// TIA Portal V20 export
TYPE "typeGlobalClockMem"
// stored: Access Published, IsFailsafeCompliant true, Namespace Safety
   STRUCT
      cycle100Msec { ExternalAccessible := 'False'; ExternalVisible := 'False'; ExternalWritable := 'False'} : Bool;   // Zeittakt 100ms / Time cycle 100ms
      cycle200Msec { ExternalAccessible := 'False'; ExternalVisible := 'False'; ExternalWritable := 'False'} : Bool;   // Zeittakt 200ms / Time cycle 200ms
      cycle400Msec { ExternalAccessible := 'False'; ExternalVisible := 'False'; ExternalWritable := 'False'} : Bool;   // Zeittakt 400ms / Time cycle 400ms
      cycle500Msec { ExternalAccessible := 'False'; ExternalVisible := 'False'; ExternalWritable := 'False'} : Bool;   // Zeittakt 500ms / Time cycle 500ms
      cycle800Msec { ExternalAccessible := 'False'; ExternalVisible := 'False'; ExternalWritable := 'False'} : Bool;   // Zeittakt 800ms / Time cycle 800ms
      cycle1000Msec { ExternalAccessible := 'False'; ExternalVisible := 'False'; ExternalWritable := 'False'} : Bool;   // Zeittakt 1,0sec / Time cycle 1,0sec
      cycle1600Msec { ExternalAccessible := 'False'; ExternalVisible := 'False'; ExternalWritable := 'False'} : Bool;   // Zeittakt 1,6sec / Time cycle 1,6sec
      cycle2000Msec { ExternalAccessible := 'False'; ExternalVisible := 'False'; ExternalWritable := 'False'} : Bool;   // Zeittakt 2,0sec / Time cycle 2,0sec
   END_STRUCT;
END_TYPE
